Staubli VAL3: getErrorCode.pgx

public program getErrorCode(num handle_, num& errorCode_[])
begin
  errorCode=errorCode[handle_]
end
